Yaskawa INFORM job: R2_W57-58-A1(80,0)AWOK.JBI

/JOB
//NAME R2_W57-58-A1(80,0)AWOK
///FOLDERNAME AWOK
//POS
///NPOS 48,48,0,3,0,0
///TOOL 0
///POSTYPE PULSE
///PULSE
C00000=107343,80978,29608,-348,54101,51738
C00001=107344,75852,40161,-399,44973,51773
C00002=107343,75531,42309,-410,43486,51780
C00003=107343,75442,43215,-414,42883,51782
C00004=107343,75365,44504,-421,42050,51786
C00005=107256,76078,45303,-339,41923,51746
C00006=107343,75365,44504,-421,42050,51786
C00007=107343,75442,43215,-414,42883,51782
C00008=107344,75475,43091,-414,42976,51782
C00009=107344,75405,44131,-419,42301,51785
C00010=107344,75475,43091,-414,42976,51782
C00011=107343,75442,43215,-414,42883,51782
C00012=107343,79315,31559,-595,72025,55971
C00013=107911,92808,47687,-889,69038,56180
C00014=107323,93257,48256,-594,68916,55978
C00015=108135,92748,47169,-1000,69330,56252
C00016=99577,100204,34867,17276,85197,57920
C00017=120731,110099,61577,-14533,111298,79491
C00018=120730,108822,63511,-14337,109508,79717
C00019=120730,108393,64390,-14262,108769,79809
C00020=120730,108506,64140,-14282,108975,79783
C00021=120730,108065,65200,-14199,108121,79888
C00022=120730,108506,64140,-14282,108975,79783
C00023=120730,108393,64390,-14262,108769,79809
C00024=120730,108719,63814,-14313,109276,79746
C00025=120730,108634,63986,-14298,109130,79764
C00026=120730,108719,63814,-14313,109276,79746
C00027=120730,108393,64390,-14262,108769,79809
C00028=120732,107903,65952,-23287,60533,68356
C00029=120732,107877,65918,-23286,60540,68355
C00030=120732,107862,65898,-23285,60544,68354
C00031=120732,107877,65918,-23286,60540,68355
C00032=120731,107909,65960,-23287,60531,68356
C00033=120731,107876,65917,-23285,60540,68354
C00034=120731,107876,65917,-23285,60540,68354
C00035=120731,107898,65946,-23287,60534,68356
C00036=147565,134559,86425,179,94382,68922
C00037=147564,133172,88551,179,92361,68918
C00038=147685,130088,85109,162,92893,68959
C00039=147595,132209,87611,175,92444,68929
C00040=147221,134171,90565,224,91636,68804
C00041=147599,129470,92489,167,88301,68900
C00042=147599,129470,92489,167,88301,68900
C00043=147589,131728,90434,175,90460,68924
C00044=147589,131728,90434,175,90460,68924
C00045=147589,135220,84634,176,95823,68932
C00046=152213,71889,2039,-9943,83128,68455
C00047=93760,62390,-25016,-9473,81706,67636
BC00000=61611,209271,1075175
BC00001=61653,209276,1075175
BC00002=65366,204356,1075175
BC00003=66851,202388,1075175
BC00004=66832,201945,1075175
BC00005=67450,201288,1075175
BC00006=66832,201945,1075175
BC00007=66851,202388,1075175
BC00008=60950,200873,1075175
BC00009=60935,200513,1075175
BC00010=60950,200873,1075175
BC00011=66851,202388,1075175
BC00012=64059,169003,1075175
BC00013=67306,165244,1075175
BC00014=67306,165244,1075175
BC00015=67306,165244,1075175
BC00016=67383,179300,1075175
BC00017=186822,178724,1075175
BC00018=188452,182222,1075175
BC00019=189104,183621,1075175
BC00020=189089,179373,1075175
BC00021=189066,178849,1075175
BC00022=189089,179373,1075175
BC00023=189104,183621,1075175
BC00024=181633,183967,1075175
BC00025=181644,186994,1075175
BC00026=181633,183967,1075175
BC00027=189104,183621,1075175
BC00028=161506,263513,998365
BC00029=161453,262432,966618
BC00030=164638,262418,966547
BC00031=161453,262432,966618
BC00032=161504,264514,1005829
BC00033=171004,262005,1020342
BC00034=169268,262194,1011548
BC00035=164921,264078,1012147
BC00036=243774,127719,1075175
BC00037=245533,128447,1075175
BC00038=245533,128447,1075175
BC00039=246236,128738,1075175
BC00040=246236,128738,1075175
BC00041=340762,208959,1075166
BC00042=340762,208959,1075166
BC00043=338632,208220,1075175
BC00044=338632,208220,1075175
BC00045=338632,208220,1075175
BC00046=338632,208220,1075175
BC00047=235674,406969,1075175
///POSTYPE ROBOT
///RECTAN
///RCONF 0,0,0,0,0,0,0,0,0,0,0,0,0,0,0,0,0,0,0,0,0,0,0,0
P00002=1043.269,21.341,-685.503,-3.2769,-33.1509,3.6066
///POSTYPE BASE
P00006=0.222,-3.123,-1.508,0.0000,0.0000,0.0000
P00022=0.222,-3.123,-1.508,0.0000,0.0000,0.0000
//INST
///DATE 2023/11/16 10:52
///ATTR SC,RW
///GROUP1 RB1,BS1
NOP
'r2_W57-58-A1(80,0)
'Path S1095
SFTOF
MOVJ C00000 BC00000 VJ=20.00
MOVJ C00001 BC00001 VJ=20.00
MOVL C00002 BC00002 V=100.0
MOVL C00003 BC00003 V=100.0
MOVL C00004 BC00004 V=60.0
REFP 3 C00005 BC00005
CALL JOB:SEARCH-R1
SET P022 P006
SFTON P022
MOVL C00006 BC00006 V=60.0
MOVL C00007 BC00007 V=100.0
MOVL C00008 BC00008 V=60.0
REFP 3 C00009 BC00009
CALL JOB:SEARCH-R1
SET P022 P006
SFTON P022
MOVL C00010 BC00010 V=60.0
MOVL C00011 BC00011 V=100.0
MOVL C00012 BC00012 V=100.0
MOVL C00013 BC00013 V=60.0
REFP 3 C00014 BC00014
CALL JOB:SEARCH-R1
SET P022 P006
SFTON P022
MOVL C00015 BC00015 V=60.0
MOVL C00016 BC00016 V=100.0
'Path S1094
COMM SFTOF
COMM MOVJ C00017 BC00017 VJ=100.00
COMM MOVL C00018 BC00018 V=400.0
COMM MOVL C00019 BC00019 V=100.0
COMM MOVL C00020 BC00020 V=60.0
COMM REFP 3 C00021 BC00021
COMM CALL JOB:SEARCH-R1
COMM SET P002 P006
COMM SFTON P002
COMM MOVL C00022 BC00022 V=60.0
COMM MOVL C00023 BC00023 V=100.0
COMM MOVL C00024 BC00024 V=60.0
COMM REFP 3 C00025 BC00025
COMM CALL JOB:SEARCH-R1
COMM SET P002 P006
COMM SFTON P002
COMM MOVL C00026 BC00026 V=60.0
COMM MOVL C00027 BC00027 V=100.0
COMM MOVL C00028 BC00028 V=100.0
COMM MOVL C00029 BC00029 V=60.0
COMM REFP 3 C00030 BC00030
COMM CALL JOB:SEARCH-R1
COMM SET P002 P006
COMM SFTON P002
COMM MOVL C00031 BC00031 V=60.0
COMM MOVL C00032 BC00032 V=100.0
COMM MOVL C00033 BC00033 V=100.0
COMM MOVL C00034 BC00034 V=400.0
COMM MOVL C00035 BC00035 V=1000.0
COMM 'Path W1084
COMM SFTOF
SFTON P022
MOVJ C00036 BC00036 VJ=20.00
MOVL C00037 BC00037 V=100.0
MOVL C00038 BC00038 V=100.0 PL=0
REFP 1 C00039 BC00039
REFP 2 C00040 BC00040
MACRO1 MJ#(0) ARGF9
ARCON
MOVL C00041 BC00041 V=11.7 ENWAIT DIS=350.0
DOUT OG#(200) 11
ARCON
MOVL C00042 BC00042 V=11.7
ARCOF
MOVL C00043 BC00043 V=100.0
MOVL C00044 BC00044 V=100.0
SFTOF
MOVJ C00045 BC00045 VJ=20.00
MOVJ C00046 BC00046 VJ=20.00
MOVJ C00047 BC00047 VJ=20.00
END
